FUNCTION_BLOCK FB_RecipeHandler
VAR_INPUT
    pSource : POINTER TO ST_Recipe;     // set by the HMI when a recipe is selected
END_VAR

METHOD Apply : BOOL
GVL_Line.stActiveRecipe := pSource^;
Apply := TRUE;
END_METHOD

END_FUNCTION_BLOCK

(* stored: Version 1.1.0.1, ProductVersion 3.1.4024.0
   POU FB_RecipeHandler: Id {1c5e16f2-3b9d-4e5b-a20c-2586b57ae556}, SpecialFunc None
   Method Apply: Id {903a5091-6983-4eed-8845-13b75b1365d9} *)
